FUNCTION FC_Setup : bool
VAR_INPUT
END_VAR
VAR
END_VAR

//READ ME FIRST////////////////////////////
///////////////////////////////////////////
//For a given machine, enable the stationEnables below for the presence of a station
//If a stationEnable is FALSE, then the related allowX below are not used

(*
General Setup Instructions
1. Follow this FC_Setup and set values TRUE/FALSE as required. Typically, only the .stationEnables can be set
2. Define the motions in the system by editing the 'MotionRowText' text list.
3. Add IO mapping and motion name text to fault messages in the system by editing the textlists in the 'X_Language Text' folder.
4. Add Power on logic
5. Add interlocks for each motion in "Sx_xx_Motion_xx_xx" PRGs in "MyAdvanceInterlock" and "MyReturnInterlock"
6. Map Inputs and outputs using "Sx_IO.Rowxx.qAdvanceCoil/Sx_IO.Rowxx.qReturnedCoil" and "Sxx_IO.Rowxx.iAdvanceDepth/Sx_IO.Rowxx.iReturnedDepth"
7. Test each motion using manual mode. Each device, e.g. a cylinder should advance and return
8. Edit other FB_HMI_Control values as required
9. Add auto logic
10. Auto Cycle --> Start
*)

//station names
//open the text list "StationNames" and edit

//setup machine
System.gSetup.stationEnable[1] := TRUE; //TRUE if station is present
System.gSetup.stationEnable[2] := FALSE; //FALSE if the station does not exist on this machine
System.gSetup.stationEnable[3] := FALSE;
System.gSetup.stationEnable[4] := FALSE;
System.gSetup.stationEnable[5] := FALSE;
System.gSetup.stationEnable[6] := FALSE;

//number of rows in each station
System.gSetup.stationFunctions[1].numRowsConfig := 9;		//18 is two pages
System.gSetup.stationFunctions[2].numRowsConfig := 9;		//9 is one page
System.gSetup.stationFunctions[3].numRowsConfig := 99;		//up to 99 rows
System.gSetup.stationFunctions[4].numRowsConfig := 99;
System.gSetup.stationFunctions[5].numRowsConfig := 99;
System.gSetup.stationFunctions[6].numRowsConfig := 99;

//set up cycle time setpoints
S1_Global.station.part.CycleTimeTarget := 60;
S1_Global.station.part.CycleTimeGrossOver := S1_Global.station.part.CycleTimeTarget  * 2;

S2_Global.station.part.CycleTimeTarget := 60;
S2_Global.station.part.CycleTimeGrossOver := S2_Global.station.part.CycleTimeTarget  * 2;

S3_Global.station.part.CycleTimeTarget := 60;
S3_Global.station.part.CycleTimeGrossOver := S3_Global.station.part.CycleTimeTarget  * 2;

S4_Global.station.part.CycleTimeTarget := 60;
S4_Global.station.part.CycleTimeGrossOver := S4_Global.station.part.CycleTimeTarget  * 2;

S5_Global.station.part.CycleTimeTarget := 60;
S5_Global.station.part.CycleTimeGrossOver := S5_Global.station.part.CycleTimeTarget  * 2;

S6_Global.station.part.CycleTimeTarget := 60;
S6_Global.station.part.CycleTimeGrossOver := S6_Global.station.part.CycleTimeTarget  * 2;

//station features
System.gSetup.stationFunctions[1].allowAutoCycle := TRUE;	//TRUE to allow auto cycle
System.gSetup.stationFunctions[1].allowManualMode := TRUE;	//Generally speaking....
System.gSetup.stationFunctions[1].allowSemiAuto := TRUE; 	//..all functions are enabled...
System.gSetup.stationFunctions[1].allowDryCycle := TRUE;	//..unless there is a good reason...
System.gSetup.stationFunctions[1].allowBypass := TRUE;		//..to disable them.
System.gSetup.stationFunctions[1].allowContinuousCycle := TRUE;
System.gSetup.stationFunctions[1].allowSingleCycle := TRUE;
System.gSetup.stationFunctions[1].allowSEOC := TRUE;
System.gSetup.stationFunctions[1].allowPowerOn := TRUE;
System.gSetup.stationFunctions[1].allowPowerOff := TRUE;
System.gSetup.stationFunctions[1].allowServicesPowerOn := TRUE;
System.gSetup.stationFunctions[1].allowRemoteControl := TRUE;
System.gSetup.stationFunctions[1].allowServicesPowerOn := TRUE;
System.gSetup.stationFunctions[1].allowSilenceHorn := TRUE;
System.gSetup.stationFunctions[1].allowGate1Req := TRUE;
System.gSetup.stationFunctions[1].allowGate2Req := TRUE;
System.gSetup.stationFunctions[1].allowLockAccessGates := TRUE;
System.gSetup.stationFunctions[1].allowEnablePendent := TRUE;


System.gSetup.stationFunctions[2].allowAutoCycle := TRUE;
System.gSetup.stationFunctions[2].allowManualMode := TRUE;
System.gSetup.stationFunctions[2].allowSemiAuto := TRUE;
System.gSetup.stationFunctions[2].allowDryCycle := TRUE;
System.gSetup.stationFunctions[2].allowBypass := TRUE;
System.gSetup.stationFunctions[2].allowContinuousCycle := TRUE;
System.gSetup.stationFunctions[2].allowSingleCycle := TRUE;
System.gSetup.stationFunctions[2].allowSEOC := TRUE;
System.gSetup.stationFunctions[2].allowPowerOn := TRUE;
System.gSetup.stationFunctions[2].allowPowerOff := TRUE;
System.gSetup.stationFunctions[2].allowServicesPowerOn := TRUE;
System.gSetup.stationFunctions[2].allowRemoteControl := TRUE;
System.gSetup.stationFunctions[2].allowServicesPowerOn := TRUE;
System.gSetup.stationFunctions[2].allowSilenceHorn := TRUE;
System.gSetup.stationFunctions[2].allowGate1Req := TRUE;
System.gSetup.stationFunctions[2].allowGate2Req := TRUE;
System.gSetup.stationFunctions[2].allowLockAccessGates := TRUE;
System.gSetup.stationFunctions[2].allowEnablePendent := TRUE;

System.gSetup.stationFunctions[3].allowAutoCycle := TRUE;
System.gSetup.stationFunctions[3].allowManualMode := TRUE;
System.gSetup.stationFunctions[3].allowSemiAuto := TRUE;
System.gSetup.stationFunctions[3].allowDryCycle := TRUE;
System.gSetup.stationFunctions[3].allowBypass := TRUE;
System.gSetup.stationFunctions[3].allowContinuousCycle := TRUE;
System.gSetup.stationFunctions[3].allowSingleCycle := TRUE;
System.gSetup.stationFunctions[3].allowSEOC := TRUE;
System.gSetup.stationFunctions[3].allowPowerOn := TRUE;
System.gSetup.stationFunctions[3].allowPowerOff := TRUE;
System.gSetup.stationFunctions[3].allowServicesPowerOn := TRUE;
System.gSetup.stationFunctions[3].allowRemoteControl := TRUE;
System.gSetup.stationFunctions[3].allowServicesPowerOn := TRUE;
System.gSetup.stationFunctions[3].allowSilenceHorn := TRUE;
System.gSetup.stationFunctions[3].allowGate1Req := TRUE;
System.gSetup.stationFunctions[3].allowGate2Req := TRUE;
System.gSetup.stationFunctions[3].allowLockAccessGates := TRUE;
System.gSetup.stationFunctions[3].allowEnablePendent := TRUE;

System.gSetup.stationFunctions[4].allowAutoCycle := TRUE;
System.gSetup.stationFunctions[4].allowManualMode := TRUE;
System.gSetup.stationFunctions[4].allowSemiAuto := TRUE;
System.gSetup.stationFunctions[4].allowDryCycle := TRUE;
System.gSetup.stationFunctions[4].allowBypass := TRUE;
System.gSetup.stationFunctions[4].allowContinuousCycle := TRUE;
System.gSetup.stationFunctions[4].allowSingleCycle := TRUE;
System.gSetup.stationFunctions[4].allowSEOC := TRUE;
System.gSetup.stationFunctions[4].allowPowerOn := TRUE;
System.gSetup.stationFunctions[4].allowPowerOff := TRUE;
System.gSetup.stationFunctions[4].allowServicesPowerOn := TRUE;
System.gSetup.stationFunctions[4].allowRemoteControl := TRUE;
System.gSetup.stationFunctions[4].allowServicesPowerOn := TRUE;
System.gSetup.stationFunctions[4].allowSilenceHorn := TRUE;
System.gSetup.stationFunctions[4].allowGate1Req := TRUE;
System.gSetup.stationFunctions[4].allowGate2Req := TRUE;
System.gSetup.stationFunctions[4].allowLockAccessGates := TRUE;
System.gSetup.stationFunctions[4].allowEnablePendent := TRUE;

System.gSetup.stationFunctions[5].allowAutoCycle := TRUE;
System.gSetup.stationFunctions[5].allowManualMode := TRUE;
System.gSetup.stationFunctions[5].allowSemiAuto := TRUE;
System.gSetup.stationFunctions[5].allowDryCycle := TRUE;
System.gSetup.stationFunctions[5].allowBypass := TRUE;
System.gSetup.stationFunctions[5].allowContinuousCycle := TRUE;
System.gSetup.stationFunctions[5].allowSingleCycle := TRUE;
System.gSetup.stationFunctions[5].allowSEOC := TRUE;
System.gSetup.stationFunctions[5].allowPowerOn := TRUE;
System.gSetup.stationFunctions[5].allowPowerOff := TRUE;
System.gSetup.stationFunctions[5].allowServicesPowerOn := TRUE;
System.gSetup.stationFunctions[5].allowRemoteControl := TRUE;
System.gSetup.stationFunctions[5].allowServicesPowerOn := TRUE;
System.gSetup.stationFunctions[5].allowSilenceHorn := TRUE;
System.gSetup.stationFunctions[5].allowGate1Req := TRUE;
System.gSetup.stationFunctions[5].allowGate2Req := TRUE;
System.gSetup.stationFunctions[5].allowLockAccessGates := TRUE;
System.gSetup.stationFunctions[5].allowEnablePendent := TRUE;

System.gSetup.stationFunctions[6].allowAutoCycle := TRUE;
System.gSetup.stationFunctions[6].allowManualMode := TRUE;
System.gSetup.stationFunctions[6].allowSemiAuto := TRUE;
System.gSetup.stationFunctions[6].allowDryCycle := TRUE;
System.gSetup.stationFunctions[6].allowBypass := TRUE;
System.gSetup.stationFunctions[6].allowContinuousCycle := TRUE;
System.gSetup.stationFunctions[6].allowSingleCycle := TRUE;
System.gSetup.stationFunctions[6].allowSEOC := TRUE;
System.gSetup.stationFunctions[6].allowPowerOn := TRUE;
System.gSetup.stationFunctions[6].allowPowerOff := TRUE;
System.gSetup.stationFunctions[6].allowServicesPowerOn := TRUE;
System.gSetup.stationFunctions[6].allowRemoteControl := TRUE;
System.gSetup.stationFunctions[6].allowServicesPowerOn := TRUE;
System.gSetup.stationFunctions[6].allowSilenceHorn := TRUE;
System.gSetup.stationFunctions[6].allowGate1Req := TRUE;
System.gSetup.stationFunctions[6].allowGate2Req := TRUE;
System.gSetup.stationFunctions[6].allowLockAccessGates := TRUE;
System.gSetup.stationFunctions[6].allowEnablePendent := TRUE;

//latch XIC messages?
S1_Global.station.Data.latchXICmsg := TRUE;
S2_Global.station.Data.latchXICmsg := FALSE;
S3_Global.station.Data.latchXICmsg := FALSE;
S4_Global.station.Data.latchXICmsg := FALSE;
S5_Global.station.Data.latchXICmsg := FALSE;
S6_Global.station.Data.latchXICmsg := FALSE;

END_FUNCTION

(* stored: Version 1.1.0.1, ProductVersion 3.1.4024.11
   POU FC_Setup: Id {054a5b72-0712-4674-ad7e-bb0ca048a77e}, SpecialFunc None *)
